FUNCTION_BLOCK EQ_LINT (* IEC 61131-3,Table 28#7 *)
  (* Standard: 61131-3 *)
  (* Version 0.1, 2006-09-14, JHC, Holobloc Inc *)
  (* Compiler header: package fb.rt.plc.comp; *)
  (* Compiler classdef: (IN1 == IN2) *)
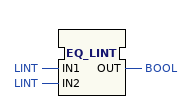
  VAR_INPUT
    IN1 : LINT;
    IN2 : LINT;
  END_VAR
  VAR_OUTPUT
    OUT : BOOL;
  END_VAR
END_FUNCTION_BLOCK
